// TIA Portal V15.1 export
// export: Created 2024-05-17T05:38:58.9837455Z, ExportSetting WithDefaults, DisplayName Totally Integrated Automation Portal, DisplayVersion V15.1 Update 5, DisplayName TIA Portal Openness, DisplayVersion V15.1 Update 5, DisplayName SINAMICS Startdrive Advanced, DisplayVersion V15.1, DisplayName G130, G150, S120, S150, SINAMICS MV, S210, DisplayVersion V15.1, DisplayName G110M, G120, G120C, G120D, G120P, DisplayVersion V15.1, DisplayName STEP 7 Professional, DisplayVersion V15.1 Update 5, DisplayName STEP 7 Safety, DisplayVersion V15.1, DisplayName WinCC Professional, DisplayVersion V15.1 Update 5, DisplayName SIMATIC Visualization Architect, DisplayVersion V15.1
FUNCTION "209230ZS01AS" : Void   // FC422, FBD
TITLE = 209230ZS01AS Panels
{ S7_Optimized_Access := 'TRUE' }
AUTHOR : VCC
VERSION : 0.1
// stored: AutoNumber false, IsIECCheckEnabled false, SetENOAutomatically False, UDAEnableTagReadback false
   VAR_OUTPUT
      O_AlarmA : Bool;   // Alarm A
      O_AlarmB : Bool;   // Alarm B
      O_AlarmC : Bool;   // Alarm C
      O_AlarmD : Bool;   // Alarm D
      O_AlarmABCondition : Bool;   // Alarm AB condition
      H_IAnim : Word;   // For animation of icon
   END_VAR
BEGIN

REGION Network 1: **** --------------------- Pushbuttons Equipment 209230AS10 --------------------- ****
END_REGION

REGION Network 2: **** 4.3 - Machine status - Operator Selection **** Pushbutton 230CA21 Buffer Conveyor to Set direction
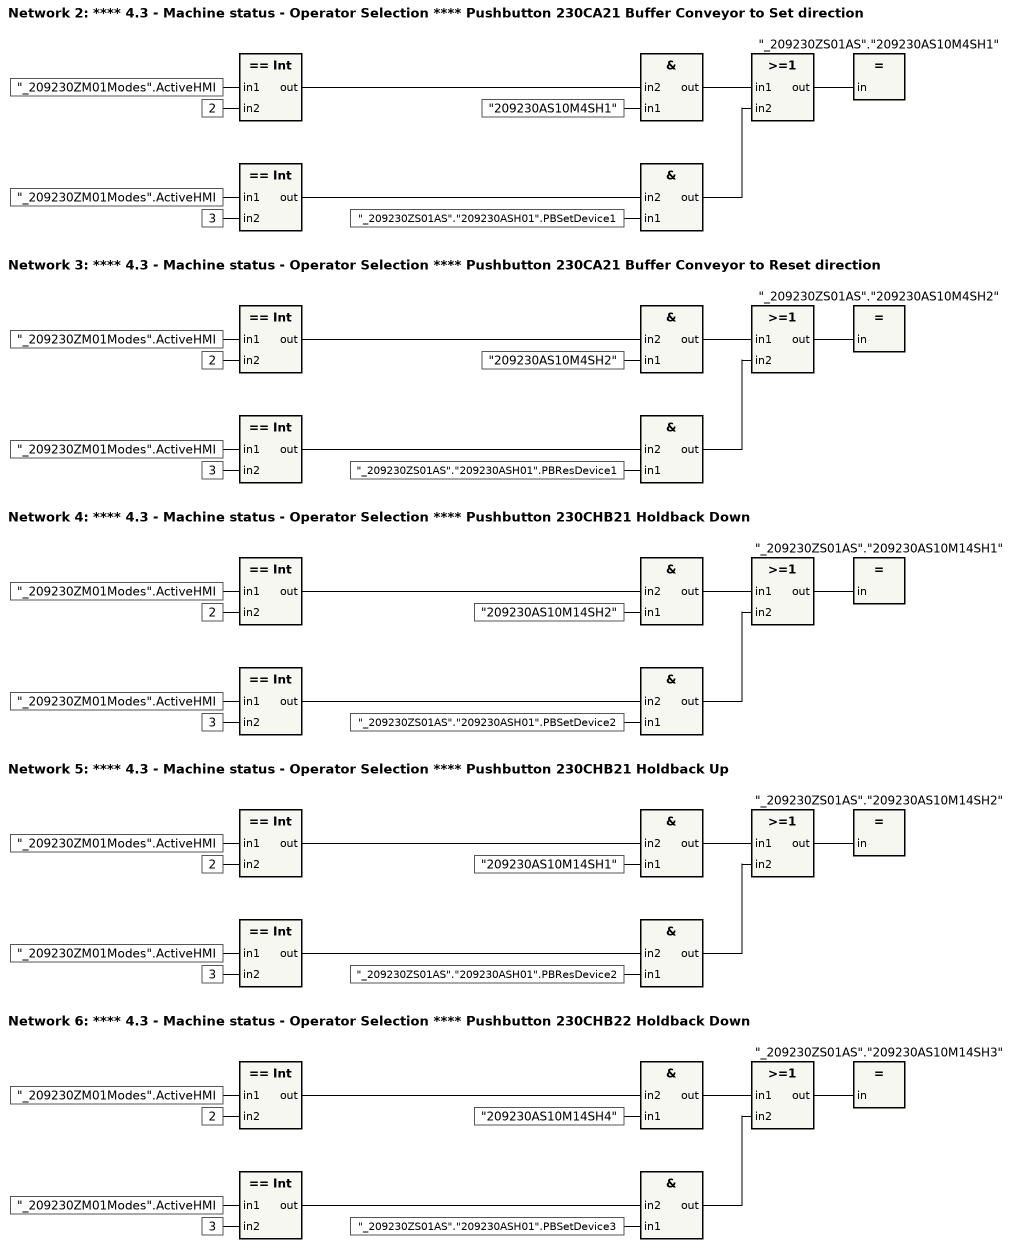
   "_209230ZS01AS"."209230AS10M4SH1" := (("_209230ZM01Modes".ActiveHMI = 2) AND "209230AS10M4SH1") OR (("_209230ZM01Modes".ActiveHMI = 3) AND "_209230ZS01AS"."209230ASH01".PBSetDevice1);
END_REGION

REGION Network 3: **** 4.3 - Machine status - Operator Selection **** Pushbutton 230CA21 Buffer Conveyor to Reset direction
   "_209230ZS01AS"."209230AS10M4SH2" := (("_209230ZM01Modes".ActiveHMI = 2) AND "209230AS10M4SH2") OR (("_209230ZM01Modes".ActiveHMI = 3) AND "_209230ZS01AS"."209230ASH01".PBResDevice1);
END_REGION

REGION Network 4: **** 4.3 - Machine status - Operator Selection **** Pushbutton 230CHB21 Holdback Down
   "_209230ZS01AS"."209230AS10M14SH1" := (("_209230ZM01Modes".ActiveHMI = 2) AND "209230AS10M14SH2") OR (("_209230ZM01Modes".ActiveHMI = 3) AND "_209230ZS01AS"."209230ASH01".PBSetDevice2);
END_REGION

REGION Network 5: **** 4.3 - Machine status - Operator Selection **** Pushbutton 230CHB21 Holdback Up
   "_209230ZS01AS"."209230AS10M14SH2" := (("_209230ZM01Modes".ActiveHMI = 2) AND "209230AS10M14SH1") OR (("_209230ZM01Modes".ActiveHMI = 3) AND "_209230ZS01AS"."209230ASH01".PBResDevice2);
END_REGION

REGION Network 6: **** 4.3 - Machine status - Operator Selection **** Pushbutton 230CHB22 Holdback Down
   "_209230ZS01AS"."209230AS10M14SH3" := (("_209230ZM01Modes".ActiveHMI = 2) AND "209230AS10M14SH4") OR (("_209230ZM01Modes".ActiveHMI = 3) AND "_209230ZS01AS"."209230ASH01".PBSetDevice3);
END_REGION

REGION Network 7: **** 4.3 - Machine status - Operator Selection **** Pushbutton 230CHB22 Holdback Up
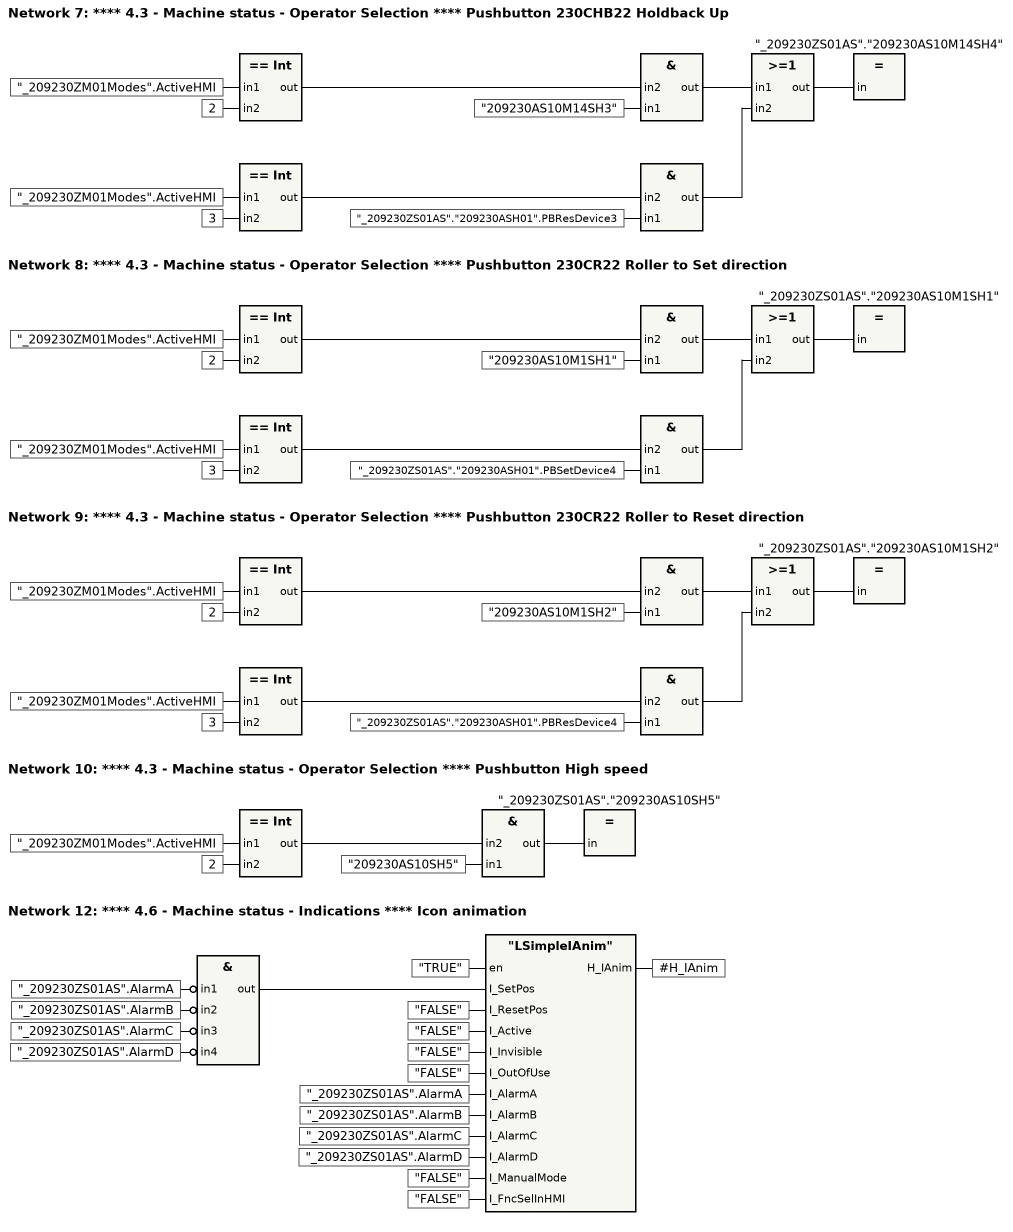
   "_209230ZS01AS"."209230AS10M14SH4" := (("_209230ZM01Modes".ActiveHMI = 2) AND "209230AS10M14SH3") OR (("_209230ZM01Modes".ActiveHMI = 3) AND "_209230ZS01AS"."209230ASH01".PBResDevice3);
END_REGION

REGION Network 8: **** 4.3 - Machine status - Operator Selection **** Pushbutton 230CR22 Roller to Set direction
   "_209230ZS01AS"."209230AS10M1SH1" := (("_209230ZM01Modes".ActiveHMI = 2) AND "209230AS10M1SH1") OR (("_209230ZM01Modes".ActiveHMI = 3) AND "_209230ZS01AS"."209230ASH01".PBSetDevice4);
END_REGION

REGION Network 9: **** 4.3 - Machine status - Operator Selection **** Pushbutton 230CR22 Roller to Reset direction
   "_209230ZS01AS"."209230AS10M1SH2" := (("_209230ZM01Modes".ActiveHMI = 2) AND "209230AS10M1SH2") OR (("_209230ZM01Modes".ActiveHMI = 3) AND "_209230ZS01AS"."209230ASH01".PBResDevice4);
END_REGION

REGION Network 10: **** 4.3 - Machine status - Operator Selection **** Pushbutton High speed
   "_209230ZS01AS"."209230AS10SH5" := ("_209230ZM01Modes".ActiveHMI = 2) AND "209230AS10SH5";
END_REGION

REGION Network 11: **** -------------------------------------------------- ****
END_REGION

REGION Network 12: **** 4.6 - Machine status - Indications **** Icon animation
   // Icon animation
   IF "TRUE" THEN
       "LSimpleIAnim"(I_SetPos := NOT "_209230ZS01AS".AlarmA AND NOT "_209230ZS01AS".AlarmB AND NOT "_209230ZS01AS".AlarmC AND NOT "_209230ZS01AS".AlarmD,
                      I_ResetPos := "FALSE",
                      I_Active := "FALSE",
                      I_Invisible := "FALSE",
                      I_OutOfUse := "FALSE",
                      I_AlarmA := "_209230ZS01AS".AlarmA,
                      I_AlarmB := "_209230ZS01AS".AlarmB,
                      I_AlarmC := "_209230ZS01AS".AlarmC,
                      I_AlarmD := "_209230ZS01AS".AlarmD,
                      I_ManualMode := "FALSE",
                      I_FncSelInHMI := "FALSE",
                      H_IAnim => #H_IAnim);
   END_IF;
END_REGION

REGION Network 13: **** 4.6 - Machine status - Indications **** Animation
   // Animation
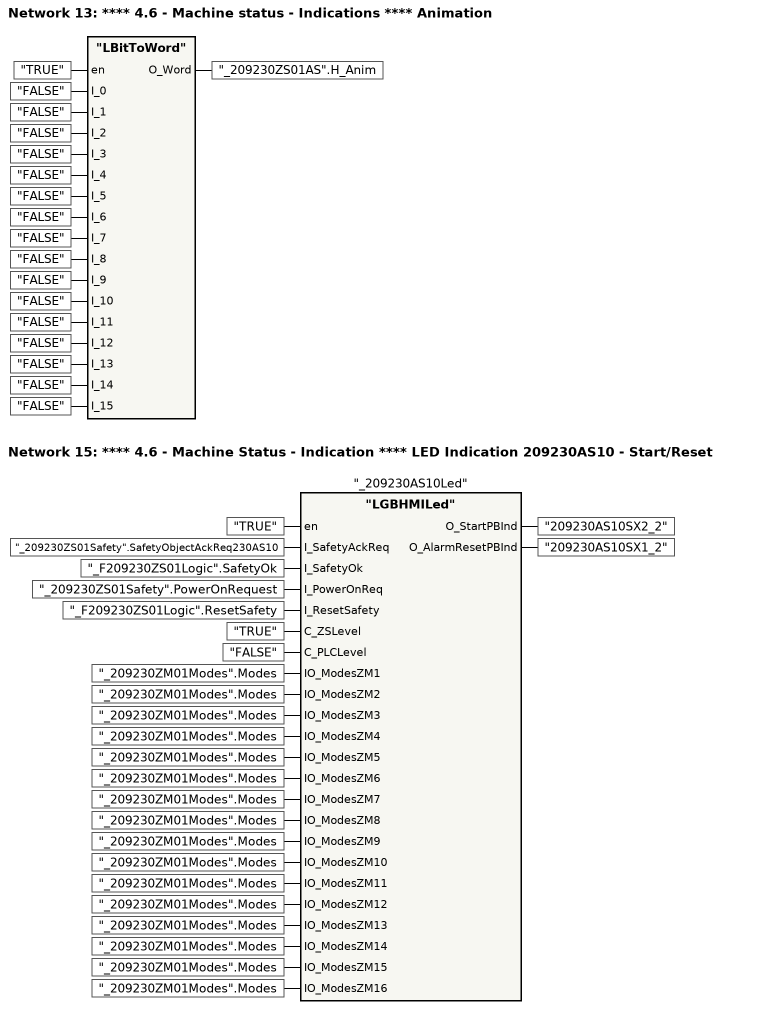
   IF "TRUE" THEN
       "LBitToWord"(I_0 := "FALSE",
                    I_1 := "FALSE",
                    I_2 := "FALSE",
                    I_3 := "FALSE",
                    I_4 := "FALSE",
                    I_5 := "FALSE",
                    I_6 := "FALSE",
                    I_7 := "FALSE",
                    I_8 := "FALSE",
                    I_9 := "FALSE",
                    I_10 := "FALSE",
                    I_11 := "FALSE",
                    I_12 := "FALSE",
                    I_13 := "FALSE",
                    I_14 := "FALSE",
                    I_15 := "FALSE",
                    O_Word => "_209230ZS01AS".H_Anim);
   END_IF;
END_REGION

NETWORK
TITLE = **** 4.6 - Machine Status - Indications **** Animation DB number
// DB number
      OPN   "_209230ZS01AS";
      L     DBNO;
      T     "_209230ZS01AS".H_DBnr;

REGION Network 15: **** 4.6 - Machine Status - Indication **** LED Indication 209230AS10 - Start/Reset
   // The Module handles indications for Start and Reset buttons
   IF "TRUE" THEN
       "_209230AS10Led"(I_SafetyAckReq := "_209230ZS01Safety".SafetyObjectAckReq230AS10,   // "LGBHMILed"
                        I_SafetyOk := "_F209230ZS01Logic".SafetyOk,
                        I_PowerOnReq := "_209230ZS01Safety".PowerOnRequest,
                        I_ResetSafety := "_F209230ZS01Logic".ResetSafety,
                        C_ZSLevel := "TRUE",
                        C_PLCLevel := "FALSE",
                        IO_ModesZM1 := "_209230ZM01Modes".Modes,
                        IO_ModesZM2 := "_209230ZM01Modes".Modes,
                        IO_ModesZM3 := "_209230ZM01Modes".Modes,
                        IO_ModesZM4 := "_209230ZM01Modes".Modes,
                        IO_ModesZM5 := "_209230ZM01Modes".Modes,
                        IO_ModesZM6 := "_209230ZM01Modes".Modes,
                        IO_ModesZM7 := "_209230ZM01Modes".Modes,
                        IO_ModesZM8 := "_209230ZM01Modes".Modes,
                        IO_ModesZM9 := "_209230ZM01Modes".Modes,
                        IO_ModesZM10 := "_209230ZM01Modes".Modes,
                        IO_ModesZM11 := "_209230ZM01Modes".Modes,
                        IO_ModesZM12 := "_209230ZM01Modes".Modes,
                        IO_ModesZM13 := "_209230ZM01Modes".Modes,
                        IO_ModesZM14 := "_209230ZM01Modes".Modes,
                        IO_ModesZM15 := "_209230ZM01Modes".Modes,
                        IO_ModesZM16 := "_209230ZM01Modes".Modes,
                        O_StartPBInd => "209230AS10SX2_2",
                        O_AlarmResetPBInd => "209230AS10SX1_2");
   END_IF;
END_REGION

REGION Network 16: **** 4.6 - Machine Status - Indication **** LED Indication 209230AS30 - Start/Reset
   // The Module handles indications for Start and Reset buttons
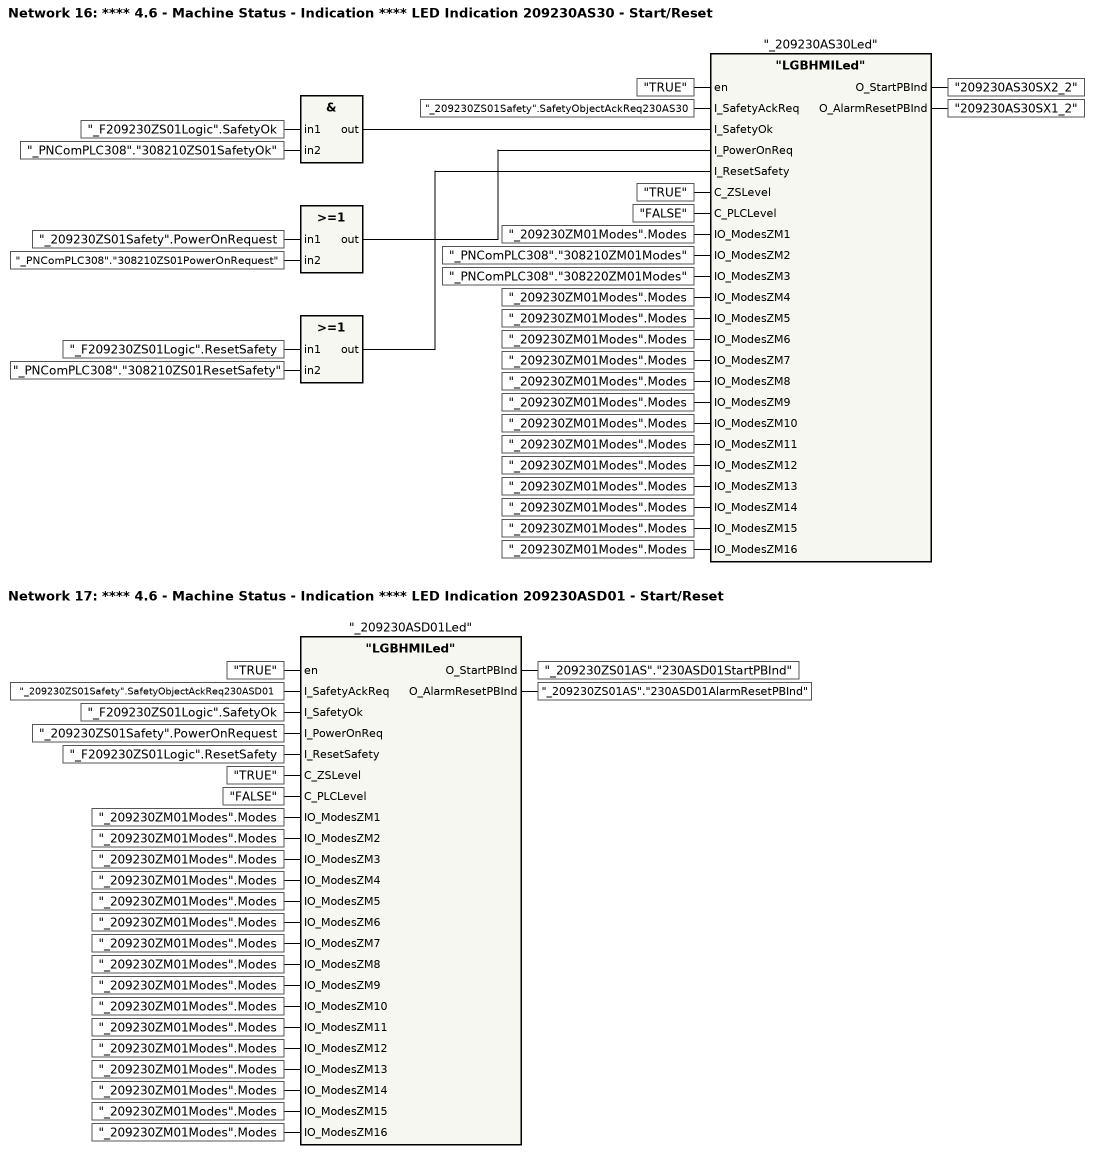
   IF "TRUE" THEN
       "_209230AS30Led"(I_SafetyAckReq := "_209230ZS01Safety".SafetyObjectAckReq230AS30,   // "LGBHMILed"
                        I_SafetyOk := "_F209230ZS01Logic".SafetyOk AND "_PNComPLC308"."308210ZS01SafetyOk",
                        I_PowerOnReq := "_209230ZS01Safety".PowerOnRequest OR "_PNComPLC308"."308210ZS01PowerOnRequest",
                        I_ResetSafety := "_F209230ZS01Logic".ResetSafety OR "_PNComPLC308"."308210ZS01ResetSafety",
                        C_ZSLevel := "TRUE",
                        C_PLCLevel := "FALSE",
                        IO_ModesZM1 := "_209230ZM01Modes".Modes,
                        IO_ModesZM2 := "_PNComPLC308"."308210ZM01Modes",
                        IO_ModesZM3 := "_PNComPLC308"."308220ZM01Modes",
                        IO_ModesZM4 := "_209230ZM01Modes".Modes,
                        IO_ModesZM5 := "_209230ZM01Modes".Modes,
                        IO_ModesZM6 := "_209230ZM01Modes".Modes,
                        IO_ModesZM7 := "_209230ZM01Modes".Modes,
                        IO_ModesZM8 := "_209230ZM01Modes".Modes,
                        IO_ModesZM9 := "_209230ZM01Modes".Modes,
                        IO_ModesZM10 := "_209230ZM01Modes".Modes,
                        IO_ModesZM11 := "_209230ZM01Modes".Modes,
                        IO_ModesZM12 := "_209230ZM01Modes".Modes,
                        IO_ModesZM13 := "_209230ZM01Modes".Modes,
                        IO_ModesZM14 := "_209230ZM01Modes".Modes,
                        IO_ModesZM15 := "_209230ZM01Modes".Modes,
                        IO_ModesZM16 := "_209230ZM01Modes".Modes,
                        O_StartPBInd => "209230AS30SX2_2",
                        O_AlarmResetPBInd => "209230AS30SX1_2");
   END_IF;
END_REGION

REGION Network 17: **** 4.6 - Machine Status - Indication **** LED Indication 209230ASD01 - Start/Reset
   // The Module handles indications for Start and Reset buttons
   IF "TRUE" THEN
       "_209230ASD01Led"(I_SafetyAckReq := "_209230ZS01Safety".SafetyObjectAckReq230ASD01,   // "LGBHMILed"
                         I_SafetyOk := "_F209230ZS01Logic".SafetyOk,
                         I_PowerOnReq := "_209230ZS01Safety".PowerOnRequest,
                         I_ResetSafety := "_F209230ZS01Logic".ResetSafety,
                         C_ZSLevel := "TRUE",
                         C_PLCLevel := "FALSE",
                         IO_ModesZM1 := "_209230ZM01Modes".Modes,
                         IO_ModesZM2 := "_209230ZM01Modes".Modes,
                         IO_ModesZM3 := "_209230ZM01Modes".Modes,
                         IO_ModesZM4 := "_209230ZM01Modes".Modes,
                         IO_ModesZM5 := "_209230ZM01Modes".Modes,
                         IO_ModesZM6 := "_209230ZM01Modes".Modes,
                         IO_ModesZM7 := "_209230ZM01Modes".Modes,
                         IO_ModesZM8 := "_209230ZM01Modes".Modes,
                         IO_ModesZM9 := "_209230ZM01Modes".Modes,
                         IO_ModesZM10 := "_209230ZM01Modes".Modes,
                         IO_ModesZM11 := "_209230ZM01Modes".Modes,
                         IO_ModesZM12 := "_209230ZM01Modes".Modes,
                         IO_ModesZM13 := "_209230ZM01Modes".Modes,
                         IO_ModesZM14 := "_209230ZM01Modes".Modes,
                         IO_ModesZM15 := "_209230ZM01Modes".Modes,
                         IO_ModesZM16 := "_209230ZM01Modes".Modes,
                         O_StartPBInd => "_209230ZS01AS"."230ASD01StartPBInd",
                         O_AlarmResetPBInd => "_209230ZS01AS"."230ASD01AlarmResetPBInd");
   END_IF;
END_REGION

REGION Network 18: **** 4.6 - Machine Status - Indication **** LED Indication 209230ASH01 - Start/Reset
   // The Module handles indications for Start and Reset buttons
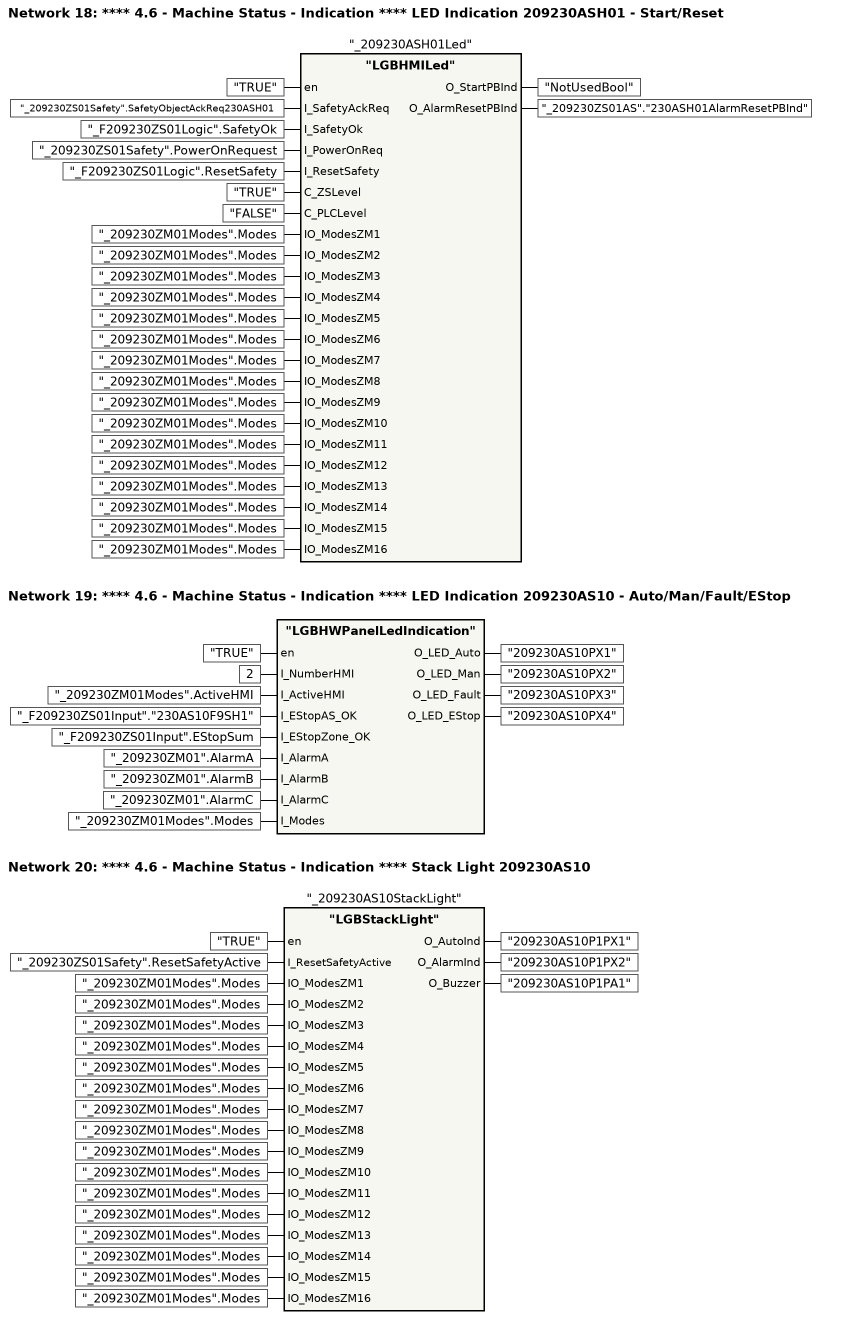
   IF "TRUE" THEN
       "_209230ASH01Led"(I_SafetyAckReq := "_209230ZS01Safety".SafetyObjectAckReq230ASH01,   // "LGBHMILed"
                         I_SafetyOk := "_F209230ZS01Logic".SafetyOk,
                         I_PowerOnReq := "_209230ZS01Safety".PowerOnRequest,
                         I_ResetSafety := "_F209230ZS01Logic".ResetSafety,
                         C_ZSLevel := "TRUE",
                         C_PLCLevel := "FALSE",
                         IO_ModesZM1 := "_209230ZM01Modes".Modes,
                         IO_ModesZM2 := "_209230ZM01Modes".Modes,
                         IO_ModesZM3 := "_209230ZM01Modes".Modes,
                         IO_ModesZM4 := "_209230ZM01Modes".Modes,
                         IO_ModesZM5 := "_209230ZM01Modes".Modes,
                         IO_ModesZM6 := "_209230ZM01Modes".Modes,
                         IO_ModesZM7 := "_209230ZM01Modes".Modes,
                         IO_ModesZM8 := "_209230ZM01Modes".Modes,
                         IO_ModesZM9 := "_209230ZM01Modes".Modes,
                         IO_ModesZM10 := "_209230ZM01Modes".Modes,
                         IO_ModesZM11 := "_209230ZM01Modes".Modes,
                         IO_ModesZM12 := "_209230ZM01Modes".Modes,
                         IO_ModesZM13 := "_209230ZM01Modes".Modes,
                         IO_ModesZM14 := "_209230ZM01Modes".Modes,
                         IO_ModesZM15 := "_209230ZM01Modes".Modes,
                         IO_ModesZM16 := "_209230ZM01Modes".Modes,
                         O_StartPBInd => "NotUsedBool",
                         O_AlarmResetPBInd => "_209230ZS01AS"."230ASH01AlarmResetPBInd");
   END_IF;
END_REGION

REGION Network 19: **** 4.6 - Machine Status - Indication **** LED Indication 209230AS10 - Auto/Man/Fault/EStop
   IF "TRUE" THEN
       "LGBHWPanelLedIndication"(I_NumberHMI := 2,
                               I_ActiveHMI := "_209230ZM01Modes".ActiveHMI,
                               I_EStopAS_OK := "_F209230ZS01Input"."230AS10F9SH1",
                               I_EStopZone_OK := "_F209230ZS01Input".EStopSum,
                               I_AlarmA := "_209230ZM01".AlarmA,
                               I_AlarmB := "_209230ZM01".AlarmB,
                               I_AlarmC := "_209230ZM01".AlarmC,
                               I_Modes := "_209230ZM01Modes".Modes,
                               O_LED_Auto => "209230AS10PX1",
                               O_LED_Man => "209230AS10PX2",
                               O_LED_Fault => "209230AS10PX3",
                               O_LED_EStop => "209230AS10PX4");
   END_IF;
END_REGION

REGION Network 20: **** 4.6 - Machine Status - Indication **** Stack Light 209230AS10
   IF "TRUE" THEN
       "_209230AS10StackLight"(I_ResetSafetyActive := "_209230ZS01Safety".ResetSafetyActive,   // "LGBStackLight"
                               IO_ModesZM1 := "_209230ZM01Modes".Modes,
                               IO_ModesZM2 := "_209230ZM01Modes".Modes,
                               IO_ModesZM3 := "_209230ZM01Modes".Modes,
                               IO_ModesZM4 := "_209230ZM01Modes".Modes,
                               IO_ModesZM5 := "_209230ZM01Modes".Modes,
                               IO_ModesZM6 := "_209230ZM01Modes".Modes,
                               IO_ModesZM7 := "_209230ZM01Modes".Modes,
                               IO_ModesZM8 := "_209230ZM01Modes".Modes,
                               IO_ModesZM9 := "_209230ZM01Modes".Modes,
                               IO_ModesZM10 := "_209230ZM01Modes".Modes,
                               IO_ModesZM11 := "_209230ZM01Modes".Modes,
                               IO_ModesZM12 := "_209230ZM01Modes".Modes,
                               IO_ModesZM13 := "_209230ZM01Modes".Modes,
                               IO_ModesZM14 := "_209230ZM01Modes".Modes,
                               IO_ModesZM15 := "_209230ZM01Modes".Modes,
                               IO_ModesZM16 := "_209230ZM01Modes".Modes,
                               O_AutoInd => "209230AS10P1PX1",
                               O_AlarmInd => "209230AS10P1PX2",
                               O_Buzzer => "209230AS10P1PA1");
   END_IF;
END_REGION

REGION Network 21: **** 7.1 - Submodule - NonMachine **** Hand Held HBA 209230ASH01
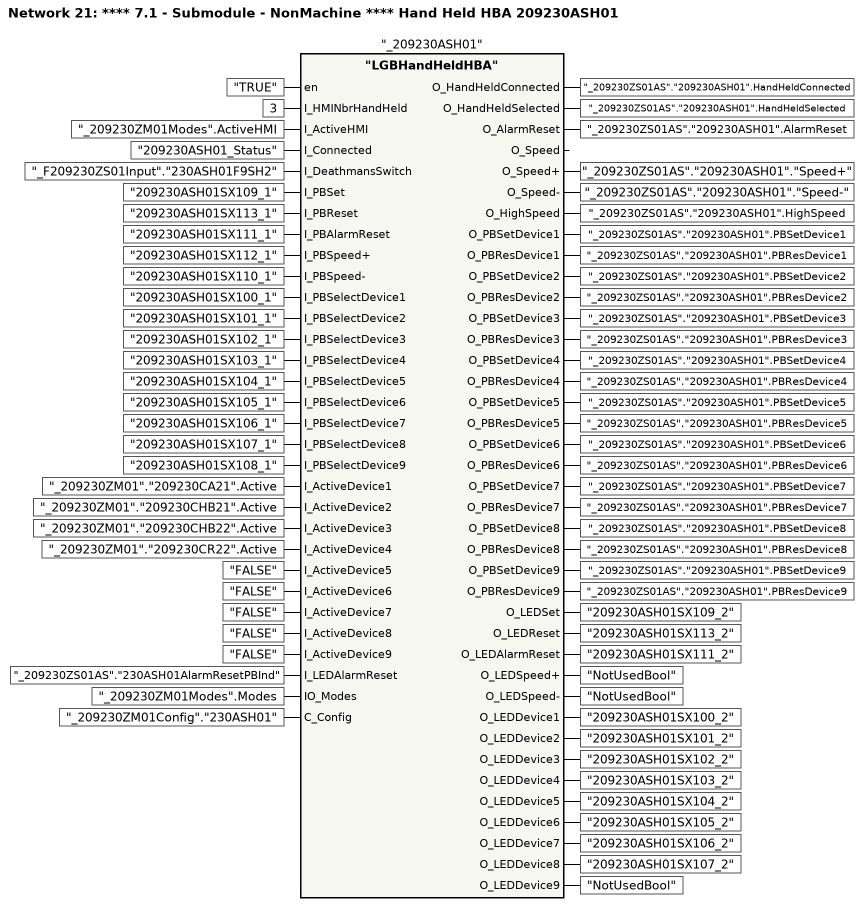
   IF "TRUE" THEN
       "_209230ASH01"(I_HMINbrHandHeld := 3,   // "LGBHandHeldHBA"
                      I_ActiveHMI := "_209230ZM01Modes".ActiveHMI,
                      I_Connected := "209230ASH01_Status",
                      I_DeathmansSwitch := "_F209230ZS01Input"."230ASH01F9SH2",
                      I_PBSet := "209230ASH01SX109_1",
                      I_PBReset := "209230ASH01SX113_1",
                      I_PBAlarmReset := "209230ASH01SX111_1",
                      "I_PBSpeed+" := "209230ASH01SX112_1",
                      "I_PBSpeed-" := "209230ASH01SX110_1",
                      I_PBSelectDevice1 := "209230ASH01SX100_1",
                      I_PBSelectDevice2 := "209230ASH01SX101_1",
                      I_PBSelectDevice3 := "209230ASH01SX102_1",
                      I_PBSelectDevice4 := "209230ASH01SX103_1",
                      I_PBSelectDevice5 := "209230ASH01SX104_1",
                      I_PBSelectDevice6 := "209230ASH01SX105_1",
                      I_PBSelectDevice7 := "209230ASH01SX106_1",
                      I_PBSelectDevice8 := "209230ASH01SX107_1",
                      I_PBSelectDevice9 := "209230ASH01SX108_1",
                      I_ActiveDevice1 := "_209230ZM01"."209230CA21".Active,
                      I_ActiveDevice2 := "_209230ZM01"."209230CHB21".Active,
                      I_ActiveDevice3 := "_209230ZM01"."209230CHB22".Active,
                      I_ActiveDevice4 := "_209230ZM01"."209230CR22".Active,
                      I_ActiveDevice5 := "FALSE",
                      I_ActiveDevice6 := "FALSE",
                      I_ActiveDevice7 := "FALSE",
                      I_ActiveDevice8 := "FALSE",
                      I_ActiveDevice9 := "FALSE",
                      I_LEDAlarmReset := "_209230ZS01AS"."230ASH01AlarmResetPBInd",
                      IO_Modes := "_209230ZM01Modes".Modes,
                      C_Config := "_209230ZM01Config"."230ASH01",
                      O_HandHeldConnected => "_209230ZS01AS"."209230ASH01".HandHeldConnected,
                      O_HandHeldSelected => "_209230ZS01AS"."209230ASH01".HandHeldSelected,
                      O_AlarmReset => "_209230ZS01AS"."209230ASH01".AlarmReset,
                      "O_Speed+" => "_209230ZS01AS"."209230ASH01"."Speed+",
                      "O_Speed-" => "_209230ZS01AS"."209230ASH01"."Speed-",
                      O_HighSpeed => "_209230ZS01AS"."209230ASH01".HighSpeed,
                      O_PBSetDevice1 => "_209230ZS01AS"."209230ASH01".PBSetDevice1,
                      O_PBResDevice1 => "_209230ZS01AS"."209230ASH01".PBResDevice1,
                      O_PBSetDevice2 => "_209230ZS01AS"."209230ASH01".PBSetDevice2,
                      O_PBResDevice2 => "_209230ZS01AS"."209230ASH01".PBResDevice2,
                      O_PBSetDevice3 => "_209230ZS01AS"."209230ASH01".PBSetDevice3,
                      O_PBResDevice3 => "_209230ZS01AS"."209230ASH01".PBResDevice3,
                      O_PBSetDevice4 => "_209230ZS01AS"."209230ASH01".PBSetDevice4,
                      O_PBResDevice4 => "_209230ZS01AS"."209230ASH01".PBResDevice4,
                      O_PBSetDevice5 => "_209230ZS01AS"."209230ASH01".PBSetDevice5,
                      O_PBResDevice5 => "_209230ZS01AS"."209230ASH01".PBResDevice5,
                      O_PBSetDevice6 => "_209230ZS01AS"."209230ASH01".PBSetDevice6,
                      O_PBResDevice6 => "_209230ZS01AS"."209230ASH01".PBResDevice6,
                      O_PBSetDevice7 => "_209230ZS01AS"."209230ASH01".PBSetDevice7,
                      O_PBResDevice7 => "_209230ZS01AS"."209230ASH01".PBResDevice7,
                      O_PBSetDevice8 => "_209230ZS01AS"."209230ASH01".PBSetDevice8,
                      O_PBResDevice8 => "_209230ZS01AS"."209230ASH01".PBResDevice8,
                      O_PBSetDevice9 => "_209230ZS01AS"."209230ASH01".PBSetDevice9,
                      O_PBResDevice9 => "_209230ZS01AS"."209230ASH01".PBResDevice9,
                      O_LEDSet => "209230ASH01SX109_2",
                      O_LEDReset => "209230ASH01SX113_2",
                      O_LEDAlarmReset => "209230ASH01SX111_2",
                      "O_LEDSpeed+" => "NotUsedBool",
                      "O_LEDSpeed-" => "NotUsedBool",
                      O_LEDDevice1 => "209230ASH01SX100_2",
                      O_LEDDevice2 => "209230ASH01SX101_2",
                      O_LEDDevice3 => "209230ASH01SX102_2",
                      O_LEDDevice4 => "209230ASH01SX103_2",
                      O_LEDDevice5 => "209230ASH01SX104_2",
                      O_LEDDevice6 => "209230ASH01SX105_2",
                      O_LEDDevice7 => "209230ASH01SX106_2",
                      O_LEDDevice8 => "209230ASH01SX107_2",
                      O_LEDDevice9 => "NotUsedBool");
   END_IF;
END_REGION

REGION Network 22: **** 8 - Outputs **** Led Indication 209230AS10 - Equipment
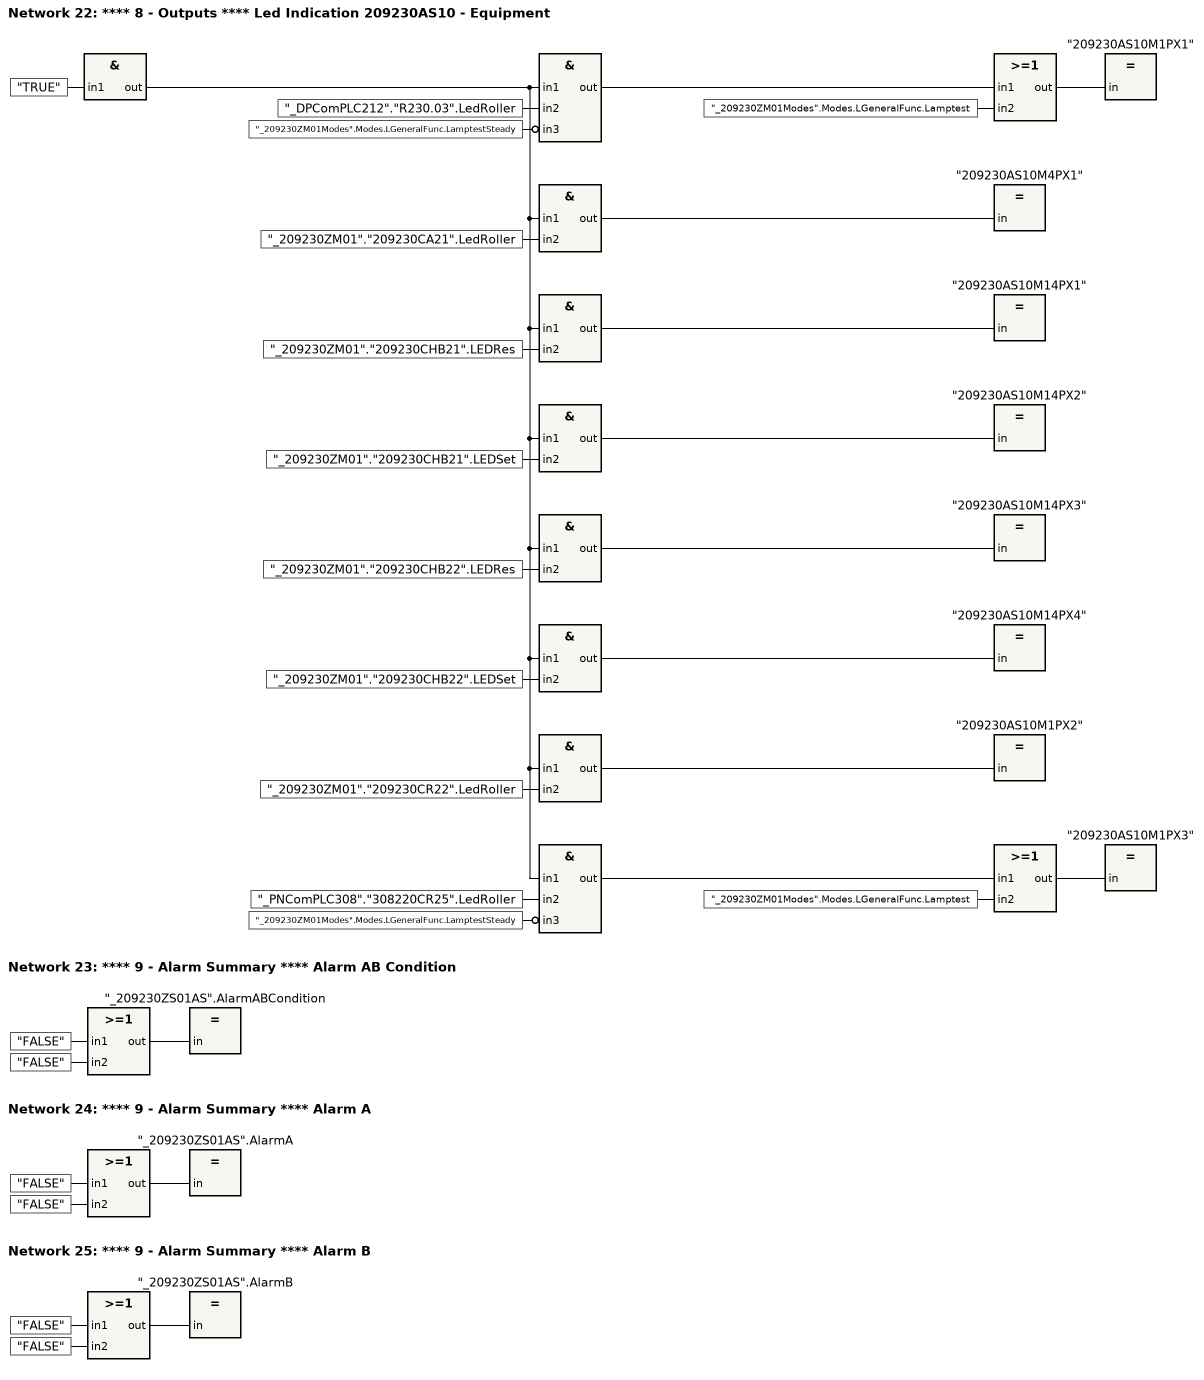
   "209230AS10M1PX1" := ("TRUE" AND "_DPComPLC212"."R230.03".LedRoller AND NOT "_209230ZM01Modes".Modes.LGeneralFunc.LamptestSteady) OR "_209230ZM01Modes".Modes.LGeneralFunc.Lamptest;
   "209230AS10M4PX1" := "TRUE" AND "_209230ZM01"."209230CA21".LedRoller;
   "209230AS10M14PX1" := "TRUE" AND "_209230ZM01"."209230CHB21".LEDRes;
   "209230AS10M14PX2" := "TRUE" AND "_209230ZM01"."209230CHB21".LEDSet;
   "209230AS10M14PX3" := "TRUE" AND "_209230ZM01"."209230CHB22".LEDRes;
   "209230AS10M14PX4" := "TRUE" AND "_209230ZM01"."209230CHB22".LEDSet;
   "209230AS10M1PX2" := "TRUE" AND "_209230ZM01"."209230CR22".LedRoller;
   "209230AS10M1PX3" := ("TRUE" AND "_PNComPLC308"."308220CR25".LedRoller AND NOT "_209230ZM01Modes".Modes.LGeneralFunc.LamptestSteady) OR "_209230ZM01Modes".Modes.LGeneralFunc.Lamptest;
END_REGION

REGION Network 23: **** 9 - Alarm Summary **** Alarm AB Condition
   // Alarm AB condition
   "_209230ZS01AS".AlarmABCondition := "FALSE" OR "FALSE";
END_REGION

REGION Network 24: **** 9 - Alarm Summary **** Alarm A
   // Summary of alarms A
   "_209230ZS01AS".AlarmA := "FALSE" OR "FALSE";
END_REGION

REGION Network 25: **** 9 - Alarm Summary **** Alarm B
   // Summary of alarms B
   "_209230ZS01AS".AlarmB := "FALSE" OR "FALSE";
END_REGION

REGION Network 26: **** 9 - Alarm Summary **** Alarm C
   // Summary of alarms C
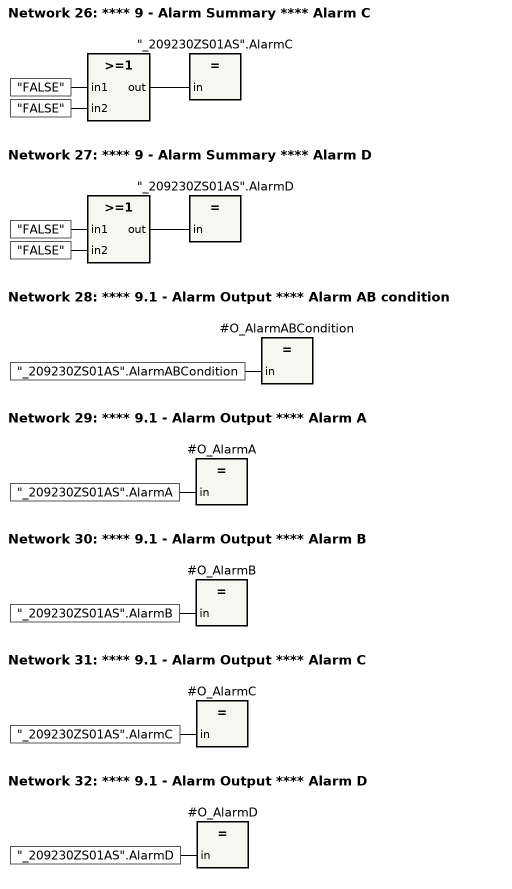
   "_209230ZS01AS".AlarmC := "FALSE" OR "FALSE";
END_REGION

REGION Network 27: **** 9 - Alarm Summary **** Alarm D
   // Summary of alarms D
   "_209230ZS01AS".AlarmD := "FALSE" OR "FALSE";
END_REGION

REGION Network 28: **** 9.1 - Alarm Output **** Alarm AB condition
   // Alarm AB condition
   #O_AlarmABCondition := "_209230ZS01AS".AlarmABCondition;
END_REGION

REGION Network 29: **** 9.1 - Alarm Output **** Alarm A
   // Output Alarm A
   #O_AlarmA := "_209230ZS01AS".AlarmA;
END_REGION

REGION Network 30: **** 9.1 - Alarm Output **** Alarm B
   // Output Alarm B
   #O_AlarmB := "_209230ZS01AS".AlarmB;
END_REGION

REGION Network 31: **** 9.1 - Alarm Output **** Alarm C
   // Output Alarm A
   #O_AlarmC := "_209230ZS01AS".AlarmC;
END_REGION

REGION Network 32: **** 9.1 - Alarm Output **** Alarm D
   // Output Alarm D
   #O_AlarmD := "_209230ZS01AS".AlarmD;
END_REGION

REGION Network 33: **** 9.2 - Alarm DWord**** Alarm To DWord
   // Alarm Word
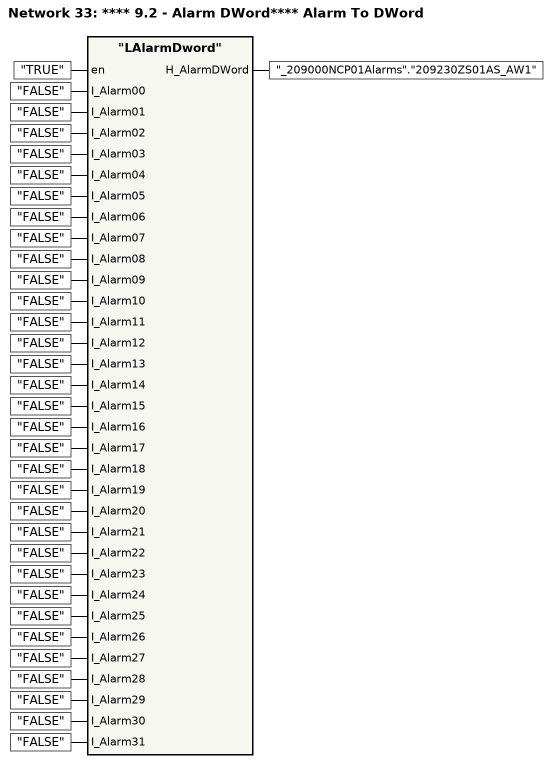
   IF "TRUE" THEN
       "LAlarmDword"(I_Alarm00 := "FALSE",
                     I_Alarm01 := "FALSE",
                     I_Alarm02 := "FALSE",
                     I_Alarm03 := "FALSE",
                     I_Alarm04 := "FALSE",
                     I_Alarm05 := "FALSE",
                     I_Alarm06 := "FALSE",
                     I_Alarm07 := "FALSE",
                     I_Alarm08 := "FALSE",
                     I_Alarm09 := "FALSE",
                     I_Alarm10 := "FALSE",
                     I_Alarm11 := "FALSE",
                     I_Alarm12 := "FALSE",
                     I_Alarm13 := "FALSE",
                     I_Alarm14 := "FALSE",
                     I_Alarm15 := "FALSE",
                     I_Alarm16 := "FALSE",
                     I_Alarm17 := "FALSE",
                     I_Alarm18 := "FALSE",
                     I_Alarm19 := "FALSE",
                     I_Alarm20 := "FALSE",
                     I_Alarm21 := "FALSE",
                     I_Alarm22 := "FALSE",
                     I_Alarm23 := "FALSE",
                     I_Alarm24 := "FALSE",
                     I_Alarm25 := "FALSE",
                     I_Alarm26 := "FALSE",
                     I_Alarm27 := "FALSE",
                     I_Alarm28 := "FALSE",
                     I_Alarm29 := "FALSE",
                     I_Alarm30 := "FALSE",
                     I_Alarm31 := "FALSE",
                     H_AlarmDWord => "_209000NCP01Alarms"."209230ZS01AS_AW1");
   END_IF;
END_REGION
END_FUNCTION
